TYPE MNG_DataArray :
ARRAY[1..MNG_BUFFER_SIZE] OF DWORD;
END_TYPE

(* stored: Version 1.1.0.1, ProductVersion 3.1.0.25
   DUT MNG_DataArray: Id {e09edf2b-4c3f-4906-ab47-a4de59dbc967} *)
